FUNCTION F_silu : lreal
VAR_INPUT
	x : LREAL;
END_VAR

F_silu := x / (1 + exp(-x));

END_FUNCTION

(* stored: Version 1.1.0.1, ProductVersion 3.1.4024.12
   POU F_silu: Id {776c6fa3-c0e3-465d-991a-a3924569a053}, SpecialFunc None *)
